// TwinCAT 3 PLC project SN001
// ProgramVersion: 3.1.4023.0
// libraries:
//   Tc2_Standard, * (Beckhoff Automation GmbH)
//   Tc2_System, * (Beckhoff Automation GmbH)
//   Tc3_Module, * (Beckhoff Automation GmbH)
// project tree:
//   / PlcTask.TcTTO
//   POUs/ FB_Test2.TcPOU, FB_TestString.TcPOU, FGetInstance.TcPOU, MAIN.TcPOU
//   POUs/Interfaces/ I_BaseString.TcIO
// real-time tasks:
//   TASK PlcTask: cycle T#10ms, priority 20, ADS port 350

CONFIGURATION SN001
    RESOURCE PLC ON TwinCAT3
        TASK PlcTask(INTERVAL := T#10ms, PRIORITY := 20);
        PROGRAM MAIN WITH PlcTask : MAIN;
    END_RESOURCE
END_CONFIGURATION

// ---- POUs/Interfaces/I_BaseString.TcIO
INTERFACE I_BaseString

METHOD GetString : STRING
VAR_INPUT
	
END_VAR
END_METHOD

END_INTERFACE

// ---- POUs/MAIN.TcPOU
PROGRAM MAIN
VAR
	fbString: FB_TestString;
	fbTest2 : FB_Test2;
	stest	: STRING;
	sTest2 	: STRING;
END_VAR




stest := FGetInstance(isample := fbString);
sTest2 := FGetInstance(isample:=fbTest2);

END_PROGRAM

// ---- POUs/FB_TestString.TcPOU
FUNCTION_BLOCK FB_TestString IMPLEMENTS I_BaseString
VAR_INPUT
END_VAR
VAR_OUTPUT
END_VAR
VAR
END_VAR

{warning 'Methodenimplementierung hinzufügen'}
METHOD GetString : STRING
 GetString := 'Test';
END_METHOD

END_FUNCTION_BLOCK

// ---- POUs/FB_Test2.TcPOU
FUNCTION_BLOCK FB_Test2 IMPLEMENTS I_BaseString
VAR_INPUT
END_VAR
VAR_OUTPUT
END_VAR
VAR
END_VAR

{warning 'Methodenimplementierung hinzufügen'}
METHOD GetString : STRING
GetString := 'Test 2';
END_METHOD

END_FUNCTION_BLOCK

// ---- POUs/FGetInstance.TcPOU
FUNCTION FGetInstance : STRING
VAR_INPUT
	isample: I_BaseString;
END_VAR
VAR
END_VAR

FGetInstance := isample.GetString();

END_FUNCTION
